# EPICS substitutions: ek9000App/Db/EL3064.substitutions
file EL3064.template
{       pattern
        {
                TERMINAL,

        }
        {
        }
}
